TYPE ST_DataSetEntry :
STRUCT
	bFlag	: BOOL;
	nValue 	: REAL;
	sMsg 	: STRING(20) := 'Unknown';
END_STRUCT
END_TYPE

(* stored: Version 1.1.0.1, ProductVersion 3.1.4024.9
   DUT ST_DataSetEntry: Id {ab4d589b-390b-4282-8bdf-faace3ec810f} *)
